FUNCTION_BLOCK ContentCollection IMPLEMENTS I_ContentCollection
VAR
	contents : Stack;
END_VAR

METHOD PUBLIC GetEnumerator : I_ForwardEnumerator
VAR_INPUT
END_VAR
GetEnumerator := contents.GetEnumerator();
END_METHOD

METHOD PUBLIC Insert
VAR_INPUT
	ContentToAdd : I_Content;
END_VAR
contents.Push(ContentToAdd);
END_METHOD

METHOD PUBLIC TryGetByName : BOOL
VAR_INPUT
	Name : STRING;
	Destination : REFERENCE TO I_Content;
END_VAR
VAR
	contentEnumerator : I_ForwardEnumerator;
	currentContent : I_Content;
END_VAR
contentEnumerator := contents.GetEnumerator();

WHILE contentEnumerator.MoveNext() DO 
	IF NOT contentEnumerator.TryGet(currentContent) THEN
		CONTINUE;
	END_IF
	
	IF currentContent.Name = Name THEN 
		TryGetByName := TRUE;
		Destination := currentContent;
		EXIT;
	END_IF

END_WHILE

contentEnumerator.Dispose();
END_METHOD

END_FUNCTION_BLOCK

(* stored: Version 1.1.0.1, ProductVersion 3.1.4024.12
   POU ContentCollection: Id {1def75d3-5565-0fe4-3612-d21a56184e52}, SpecialFunc None
   Method GetEnumerator: Id {019ffe09-1fd9-0e51-1027-51f2c74291ce}
   Method Insert: Id {648c5496-cfa7-07d8-3d0d-c88b3dcf6ad3}
   Method TryGetByName: Id {edbb8fd1-89ca-0968-2295-bfb960669b42} *)
